// TIA Portal V19 export
FUNCTION_BLOCK "FB_CM_Cilinder"   // FB1, FBD
TITLE = FB_CM_Cilinder AP BIB
{ S7_Optimized_Access := 'FALSE' }
// stored: SetENOAutomatically false
   VAR_INPUT
      iMode_Aut : Bool;
      iCmd_Aut_Out : Bool;
      iCmd_Aut_In : Bool;
      iCmd_Man_Out : Bool;
      iCmd_Man_In : Bool;
      iIntLock_Out : Bool;
      iIntLock_In : Bool;
      iSetting_Alm_Fb_En : Bool;
      iSen_Fb_Out : Bool;
      iSen_Fb_In : Bool;
      iCmd_Reset_Alm : Bool;
      iSetting_Alm_Fb_Time : Time;
   END_VAR
   VAR_OUTPUT
      oOut : Bool;
      oIn : Bool;
      oAlm_Fb_Out : Bool;
      oAlm_Fb_In : Bool;
   END_VAR
   VAR
      sHulpM : Array[0..15] of Bool;
      IEC_Timer_0_Instance { S7_SetPoint := 'True'} : TON_TIME;
      IEC_Timer_0_Instance_2 { S7_SetPoint := 'True'} : TON_TIME;
      s_iCmd_Auto_Out { S7_SetPoint := 'True'} : Bool;
      s_iCmd_Auto_In : Bool;
      s_iCmd_Man_Out_TRIG : Bool;
      s_iCmd_Man_In_TRIG : Bool;
   END_VAR
   VAR_TEMP   // added for the SCL form of the ladder/FBD networks
      _w1 : Bool;
   END_VAR
BEGIN

REGION Network 1: check input cmds in combination with mode and interlock
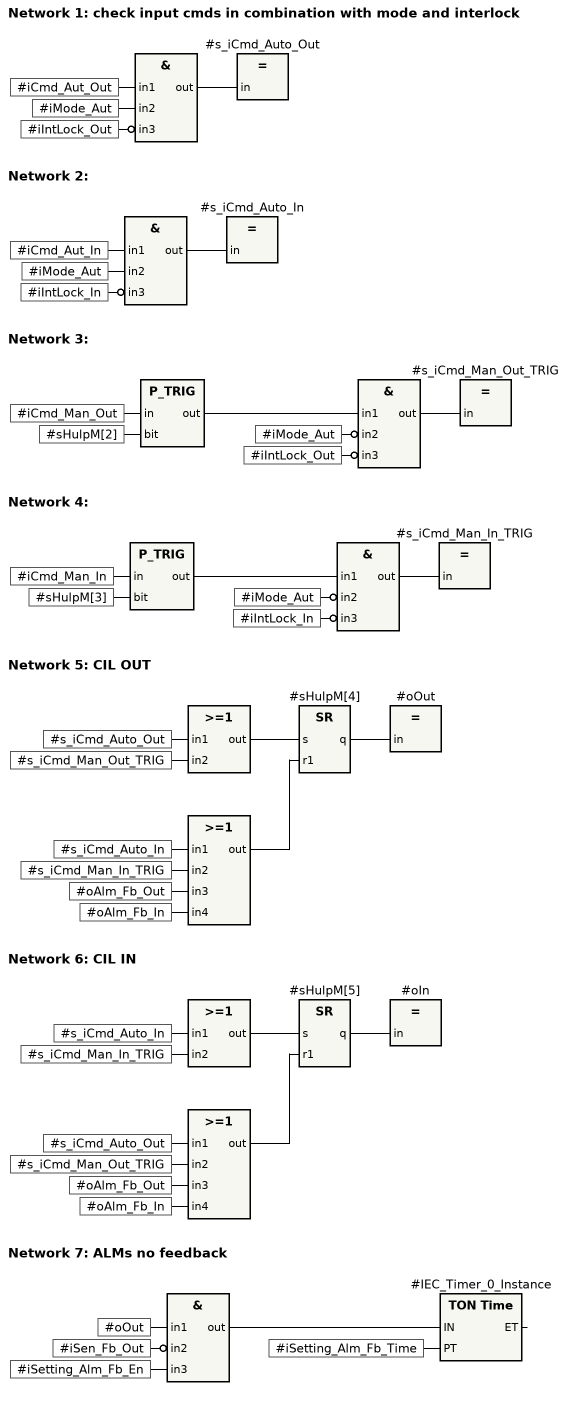
   #s_iCmd_Auto_Out := #iCmd_Aut_Out AND #iMode_Aut AND NOT #iIntLock_Out;
END_REGION

REGION Network 2
   #s_iCmd_Auto_In := #iCmd_Aut_In AND #iMode_Aut AND NOT #iIntLock_In;
END_REGION

REGION Network 3
   #_w1 := #iCmd_Man_Out AND NOT #sHulpM[2];   // rising edge
   #sHulpM[2] := #iCmd_Man_Out;
   #s_iCmd_Man_Out_TRIG := #_w1 AND NOT #iMode_Aut AND NOT #iIntLock_Out;
END_REGION

REGION Network 4
   #_w1 := #iCmd_Man_In AND NOT #sHulpM[3];   // rising edge
   #sHulpM[3] := #iCmd_Man_In;
   #s_iCmd_Man_In_TRIG := #_w1 AND NOT #iMode_Aut AND NOT #iIntLock_In;
END_REGION

REGION Network 5: CIL OUT
   // SET cilinder out: auto or man out command
   // 
   // RESET cilinder out: auto or man in command or alarm
   IF #s_iCmd_Auto_Out OR #s_iCmd_Man_Out_TRIG THEN
       #sHulpM[4] := TRUE;   // SR flip-flop
   END_IF;
   IF #s_iCmd_Auto_In OR #s_iCmd_Man_In_TRIG OR #oAlm_Fb_Out OR #oAlm_Fb_In THEN #sHulpM[4] := FALSE; END_IF;
   #oOut := #sHulpM[4];
END_REGION

REGION Network 6: CIL IN
   // SET cilinder in: auto or man in command
   // 
   // RESET cilinder in: auto or man out command or alarm
   IF #s_iCmd_Auto_In OR #s_iCmd_Man_In_TRIG THEN
       #sHulpM[5] := TRUE;   // SR flip-flop
   END_IF;
   IF #s_iCmd_Auto_Out OR #s_iCmd_Man_Out_TRIG OR #oAlm_Fb_Out OR #oAlm_Fb_In THEN
       #sHulpM[5] := FALSE;
   END_IF;
   #oIn := #sHulpM[5];
END_REGION

REGION Network 7: ALMs no feedback
   #IEC_Timer_0_Instance(IN := #oOut AND NOT #iSen_Fb_Out AND #iSetting_Alm_Fb_En, PT := #iSetting_Alm_Fb_Time);   // TON
END_REGION

REGION Network 8
   // om compatibel te zijn met 300-PLC, mag er niets achter de TON worden geprogrammeerd
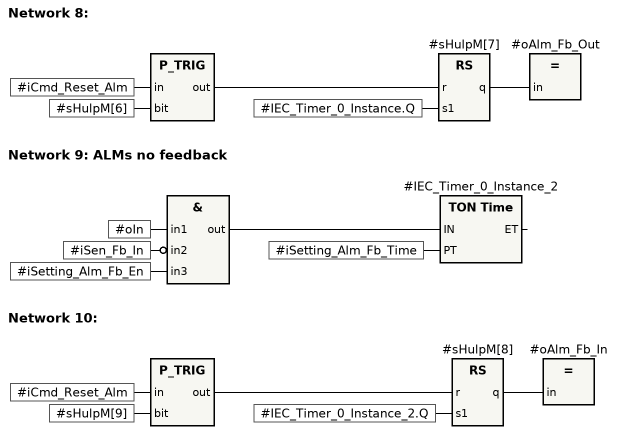
   #_w1 := #iCmd_Reset_Alm AND NOT #sHulpM[6];   // rising edge
   #sHulpM[6] := #iCmd_Reset_Alm;
   IF #_w1 THEN
       #sHulpM[7] := FALSE;   // RS flip-flop
   END_IF;
   IF #IEC_Timer_0_Instance.Q THEN #sHulpM[7] := TRUE; END_IF;
   #oAlm_Fb_Out := #sHulpM[7];
END_REGION

REGION Network 9: ALMs no feedback
   #IEC_Timer_0_Instance_2(IN := #oIn AND NOT #iSen_Fb_In AND #iSetting_Alm_Fb_En, PT := #iSetting_Alm_Fb_Time);   // TON
END_REGION

REGION Network 10
   #_w1 := #iCmd_Reset_Alm AND NOT #sHulpM[9];   // rising edge
   #sHulpM[9] := #iCmd_Reset_Alm;
   IF #_w1 THEN
       #sHulpM[8] := FALSE;   // RS flip-flop
   END_IF;
   IF #IEC_Timer_0_Instance_2.Q THEN #sHulpM[8] := TRUE; END_IF;
   #oAlm_Fb_In := #sHulpM[8];
END_REGION

REGION Network 11: statusword TODO
END_REGION
END_FUNCTION_BLOCK
